FUNCTION_BLOCK FB_Obj_Error_Schrauber
VAR_INPUT

	I_fbFehlerNachladen						:FB_ErrorCnt;	(* Fehler Nachladen, Schraube fehlt *)
	I_fbFehlerLangsameGeschwindigkeit	:FB_ErrorCnt;	(* Langsame Geschwindigkeit wird nicht erreicht *)
	I_fbFehlerTiefeSolldrehzahl			:FB_ErrorCnt;	(* Schraubtiefe für Solldrehzahl wird nicht erreicht *)
	I_fbFehler_Tiefe							:FB_ErrorCnt;	(* Tiefe nicht erreicht *)
	I_fbFehler_Tiefe2							:FB_ErrorCnt;	(* Tiefe nicht erreicht, obwohl Schrauber dreht *)
	I_fbFehler_TiefeUeberschritten		:FB_ErrorCnt;	(* Tiefe überschritten *)
	I_fbFehler_Sollmoment					:FB_ErrorCnt;	(* Drehmoment nicht erreicht*)
	I_fbFehler_Schrauberstange				:FB_ErrorCnt;	(* Fehler beim heben/senken der Schrauberstange *)
	I_fbFehlerAuswurf							:FB_ErrorCnt;	(* Fehler beim Auswerfen *)
	I_sStatus									:STRING;

END_VAR
VAR_OUTPUT
END_VAR
VAR
END_VAR

;

END_FUNCTION_BLOCK

(* stored: Version 1.1.0.1, ProductVersion 3.1.4024.12
   POU FB_Obj_Error_Schrauber: Id {418c98f1-700e-44c2-9128-439532005530}, SpecialFunc None *)
